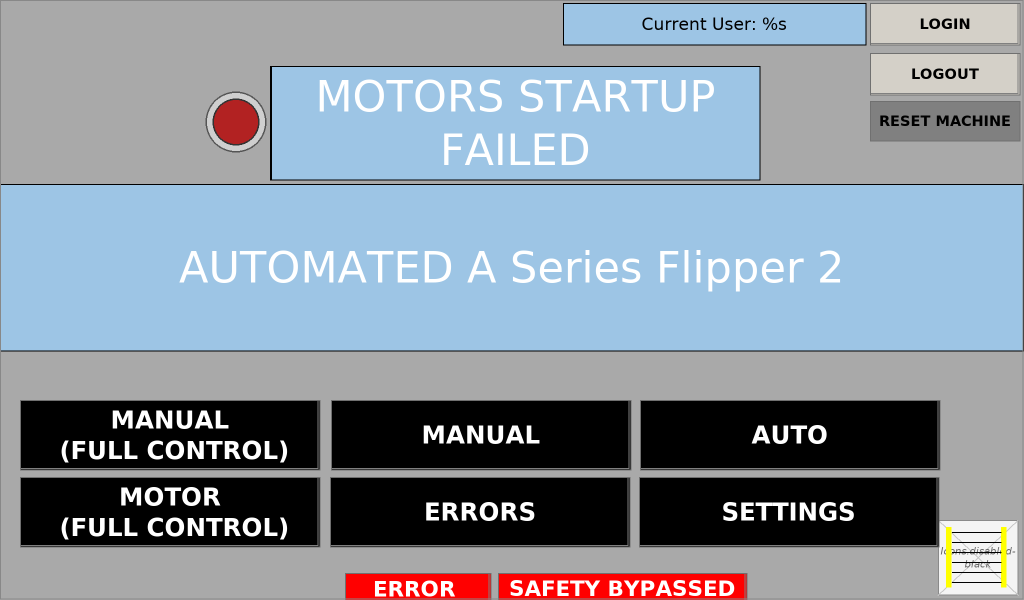
VISUALIZATION mainScreen  // 1024x600
    Image (938,520 80x75), invisible if: MAIN.bHideLtCurtainDisable, image: Icons.disabled-black
    Textfield (0,184 1024x167), "AUTOMATED A Series Flipper 2"
    Button (331,400 300x70), "MANUAL", invisible if: NOT GVL_machine.bMotorsInitialized
        OnMouseClick: change screen: manualScreen
        OnMouseClick: execute { GVL_machine.nPageIndex := 5; }
    Button (640,400 300x70), "AUTO", invisible if: NOT GVL_machine.bMotorsInitialized
        OnMouseClick: change screen: eflexScreen
        OnMouseClick: execute { GVL_machine.nPageIndex := 10; }
    Button (870,3 150x42), "LOGIN"
        OnMouseDown: VisuUserMgmt Type=Login
    Button (870,53 150x42), "LOGOUT"
        OnMouseDown: VisuUserMgmt Type=Logout
    Group (946,527 60x60), invisible if: GVL_machine.bSafetyBypass
        toggle GVL_machine.bMuteSafety
        Rectangle (0,0 5x60)
        Rectangle (55,0 5x60)
        Line (6,5) (55,5)
        Line (6,15) (55,15)
        Line (6,25) (55,25)
        Line (6,35) (55,35)
        Line (6,45) (55,45)
        Line (6,55) (55,55)
    Lamp1 (201,87 70x70), variable: NOT GVL_machine.bMotorsInitialized, invisible if: GVL_machine.bMotorsInitialized, style: Lamp-Lamp1-Red
    Textfield (270,66 489x114), "MOTORS STARTUP Please wait...", invisible if: GVL_machine.bMotorsInitialized
    Textfield (271,66 489x114), "MOTORS STARTUP FAILED", invisible if: NOT GVL_machine.bMotorInitFailedDisp
    Button (498,573 249x31), "SAFETY BYPASSED", invisible if: NOT GVL_machine.bSafetyBypass
        OnMouseDown: change screen: safetyDisableWarning
    Button (330,477 300x70), "ERRORS", invisible if: NOT GVL_machine.bMotorsInitialized
        OnMouseClick: change screen: errorScreen
    Button (639,477 300x70), "SETTINGS", invisible if: NOT GVL_machine.bMotorsInitialized
        OnMouseClick: change screen: settingsScreen
    Button (345,573 146x32), "ERROR", invisible if: NOT GVL_machine.bDispErrorIcon
        OnMouseDown: change screen: errorScreen
    Button (20,400 300x70), "MANUAL (FULL CONTROL)", invisible if: NOT GVL_machine.bMotorsInitialized
        OnMouseClick: change screen: manualBypassedScreen
        OnMouseClick: execute { GVL_machine.nPageIndex := 5; }
    Textfield (563,3 303x42), "Current User: %s", text variable: VisuElems.CurrentUserName
    Button (870,101 150x40), "RESET MACHINE"
        OnMouseDown: toggle GVL_machine.bResetMachine
    Button (20,477 300x70), "MOTOR (FULL CONTROL)", invisible if: NOT GVL_machine.bMotorsInitialized
        OnMouseClick: change screen: multiControlScreen
        OnMouseClick: execute { GVL_machine.nPageIndex := 20; }
END_VISUALIZATION

(* stored: Version 1.1.0.1, ProductVersion 3.1.4024.15
   Visu mainScreen: Id {38e0b119-67a0-4a4d-bbd0-34c620d1c795} *)
